(* CoDeSys 2.3.9.35 project: 01_fb_debounce.pro *)
(* Libraries: Standard.LIB 4.10.05 11:14:46 *)

(* POU PLC_PRG, ST *)
PROGRAM PLC_PRG
VAR
	Button		:		BOOL;
	LED			:		BOOL;
	Debounce		:		FB_Debounce;
END_VAR
Debounce(InputToDebounce:= Button, DebounceTime:= 2000, FB_Enable:= TRUE, DebouncedInput=> );

IF Debounce.DebouncedInput THEN
	LED := TRUE;
ELSE
	LED := FALSE;
END_IF;
END_PROGRAM

(* POU FB_Debounce, ST *)
FUNCTION_BLOCK FB_Debounce

(*	This FUNCTION block filters unstable digital input transitions using a debounce logic.
	If the input changes, a timer is activated.
	The output updates only if the input remains stable for the debounce period.
	Bu fonksiyon bloğu, kararsız dijital giriş GEçişlerini bir debounce mantığı ile filtreler.
	Giriş değiştiğinde bir zamanlayıcı başlatılır ve giriş belirlenen süre boyunca kararlı kalırsa çıkış güncellenir. *)

VAR_INPUT
	InputToDebounce	: BOOL;						(* Input Before Debounce - Filtreleme Öncesi Giriş *)
	DebounceTime		: INT;						(* Debounce Time In Milliseconds - Filtreleme Süresi (Milisaniye) *)
	FB_Enable			: BOOL;						(* Function Block Enable - Fonksiyon Bloğu Etkinleştirme *)
END_VAR

VAR_OUTPUT
	DebouncedInput		: BOOL;						(* Input After Debounce - Filtreleme Sonrası Giriş *)
END_VAR

VAR
	DebounceTimer		: TON;	  					(* Timer for Debouncing - Filtreleme için Zamanlayıcı *)
	LastState			: BOOL;						(* Last Stable State - Son Kararlı Durum*)
	InputChanged		: BOOL;						(* lag for Change in Input - Giriş Değişim Bayrağı *)
END_VAR
(* Last Stable State - Son Kararlı Durum*)
LastState := InputToDebounce;

(* Start Debouncing If Enable is Active - Enable Girişi Aktifse Filtreleme İşlemine Başla *)
IF (FB_Enable) THEN
	(* Check IF Input Changed - Giriş Değişti Mi Kontrol Et *)
	InputChanged := (InputToDebounce <> LastState);

	(* Timer Initialization *)
	DebounceTimer(IN := InputChanged, PT := INT_TO_TIME(DebounceTime));

	(* Update the Output If Input is Stable - Giriş Kararlıysa Çıkışı Güncelle *)
	IF DebounceTimer.Q THEN
		DebouncedInput := InputToDebounce;
		LastState := InputToDebounce;
	(* Do Not Update the Output If Input is Unstable - Giriş Kararsızsa Çıkışı Güncelleme *)
	ELSE
		DebouncedInput := LastState;
	END_IF
(* Do Nothing If Enable is Inactive - Enable Girişi Aktif Değilse Birşey Yapma *)
END_IF
END_FUNCTION_BLOCK
